Yaskawa INFORM job: FMTV_HOOD_GRILL.JBI

/JOB
//NAME FMTV_HOOD_GRILL
//POS
///NPOS 94,0,0,0,0,0
///TOOL 0
///POSTYPE PULSE
///PULSE
C00000=-47368,-58389,-75463,-75325,82045,-91552
C00001=-47476,-117254,-81462,-92967,88282,-121381
C00002=-47585,-150180,-39020,-110955,95029,-145196
C00003=-23270,-163326,-19972,-112032,80023,-131681
C00004=-25712,-159380,-18293,-113523,79114,-132193
C00005=-33335,-143978,-10206,-123508,65501,-132940
C00006=-42763,-128241,194,-135326,52037,-131772
C00007=-34360,-122011,4195,-131468,51961,-132252
C00008=23040,-127606,-726,-98184,56131,-134608
C00009=54530,-133930,-312,-87484,54655,-130791
C00010=68015,-137434,2378,-86925,51565,-126975
C00011=68015,-137434,2378,-86925,51565,-126975
C00012=70681,-138644,2888,-85845,52080,-126328
C00013=71040,-140703,2447,-86259,52088,-125743
C00014=69846,-144743,783,-88040,51792,-124880
C00015=57718,-148947,-5081,-83684,62309,-128964
C00016=53995,-150636,-6769,-82722,66165,-129759
C00017=48232,-153207,-9364,-79812,75001,-130904
C00018=44695,-155503,-11225,-75321,85283,-131266
C00019=36329,-165923,-20799,-76940,81382,-133395
C00020=32510,-169572,-22983,-79666,80545,-133049
C00021=-44932,-162730,-9861,-129768,80460,-128201
C00022=-46663,-160332,-8884,-130899,79792,-128432
C00023=-49044,-157772,-7071,-132541,79251,-128470
C00024=-34601,-158442,-13610,-121844,79482,-130617
C00025=-34196,-157366,-13562,-121475,79274,-130894
C00026=-74927,-119102,15325,-149774,69260,-130968
C00027=-88106,-120838,19729,-158428,69500,-128950
C00028=-97244,-122496,24507,-164049,70779,-127710
C00029=-62772,-164018,-8236,-136847,75645,-129302
C00030=-22020,-164296,-20741,-110455,80031,-133645
C00031=-23986,-161695,-19560,-112089,79534,-132888
C00032=-25743,-159215,-18122,-113544,79109,-132191
C00033=7628,-162474,-22830,-93471,80813,-134336
C00034=38278,-166162,-20603,-75650,81675,-133226
C00035=48223,-172527,-17821,-220718,66953,-61657
C00036=20447,-173972,-28067,-239715,62384,-67258
C00037=18257,-169178,-23297,-241360,62687,-67091
C00038=19966,-167669,-22486,-240275,62232,-66992
C00039=54812,-127092,1429,-219590,50281,-66184
C00040=53722,-119295,5623,-221586,49019,-65115
C00041=3138,-117684,4029,-257945,62693,-59441
C00042=-54590,-119527,6471,-291312,81310,-61600
C00043=-61303,-121629,6130,-295408,82823,-62492
C00044=-62473,-124760,4446,-296058,82813,-62956
C00045=-61383,-127382,2761,-295300,82324,-63140
C00046=-45291,-158436,-14199,-283363,76411,-66448
C00047=-36803,-168530,-21385,-279249,73403,-67202
C00048=-33637,-169122,-22414,-277154,72885,-67040
C00049=-8268,-168152,-25177,-260735,67443,-65637
C00050=19974,-167686,-22517,-240273,62227,-66989
C00051=27011,-166914,-18516,-232160,63405,-68805
C00052=41789,-166510,-12245,-220087,63923,-71032
C00053=36873,-171047,-15710,-223565,64778,-70981
C00054=-30875,-170872,-20008,-275129,71015,-67437
C00055=-28839,-166908,-10700,-269968,72597,-69697
C00056=-24201,-165834,-10805,-266909,72004,-69362
C00057=15715,-164670,-9145,-238305,67431,-70401
C00058=16294,-164883,-9077,-237836,67450,-70496
C00059=15032,-168908,-9930,-238193,68465,-71268
C00060=-16532,-170220,-12590,-261050,71283,-70207
C00061=-22086,-169030,-11677,-265035,71861,-70073
C00062=-25053,-166420,-10957,-267434,72126,-69490
C00063=-28592,-172919,-21943,-270605,72527,-68220
C00064=22123,-170087,-18028,-234219,65785,-69866
C00065=20623,-164258,-8108,-234618,67125,-70753
C00066=23795,-164163,-6635,-232067,67258,-71214
C00067=37423,-164557,-4674,-225452,64295,-71455
C00068=49664,-167838,-5549,-221136,60772,-72368
C00069=50042,-168090,-5420,-220785,60902,-72462
C00070=48310,-171489,-6267,-221593,61991,-72941
C00071=47370,-171605,-6665,-222333,61921,-72856
C00072=34595,-170073,-7542,-227989,64921,-72953
C00073=21833,-169684,-9235,-234274,67927,-72789
C00074=20032,-169188,-9766,-235757,67758,-72479
C00075=22853,-164534,-7043,-232761,67333,-71170
C00076=19415,-164420,-8530,-235544,67166,-70642
C00077=23719,-173498,-25771,-233839,64304,-68922
C00078=56681,-170652,-7579,-211590,63873,-72674
C00079=53657,-165861,834,-213371,65473,-73133
C00080=55028,-166339,2357,-212686,65788,-74745
C00081=76216,-161231,29355,-196807,75399,-75518
C00082=76318,-160276,31966,-195629,77283,-75776
C00083=75919,-161073,31738,-195883,77558,-75842
C00084=71583,-166800,24804,-195873,73324,-78712
C00085=69455,-168811,22349,-196597,72549,-80310
C00086=67389,-170127,19199,-198092,71648,-80274
C00087=49281,-173575,-1247,-212167,63667,-78545
C00088=49088,-172813,-1584,-212451,63187,-78362
C00089=54651,-166467,2917,-212327,66600,-74972
C00090=59119,-174402,-10513,-209681,64182,-74287
C00091=59119,-174402,-10513,-209681,64182,-74287
C00092=-41638,-117344,-74516,-143224,92250,-82798
C00093=-47368,-58389,-75463,-75325,82045,-91552
//INST
///DATE 2023/03/28 17:51
///ATTR SC,RW
///GROUP1 RB1
NOP
MOVJ C00000 VJ=65.00  //SAW CHANGE
MOVJ C00001 VJ=65.00  //OVER RIB
MOVJ C00002 VJ=65.00  //ROTATE TO SQUARE UP
MOVJ C00003 VJ=65.00  //ABOVE CUT
MOVL C00004 V=30.0  //INTO CUT
MOVL C00005 V=30.0
MOVL C00006 V=30.0  //BOTTOM INSIDE CORNER
MOVL C00007 V=30.0  //END OF ANGLE
MOVL C00008 V=30.0
MOVL C00009 V=30.0
MOVL C00010 V=30.0
MOVC C00011 V=30.0
MOVC C00012 V=30.0
MOVC C00013 V=30.0
MOVC C00014 V=30.0
MOVL C00015 V=30.0
MOVL C00016 V=30.0
MOVL C00017 V=30.0
MOVL C00018 V=30.0
MOVL C00019 V=30.0
MOVL C00020 V=45.0  //AWAY FROM CUT
MOVL C00021 V=65.0  //UP TO CENTER
MOVL C00022 V=15.0
MOVL C00023 V=15.0  //INTO CENTER
MOVL C00024 V=30.0  //RIGHT TOP CORNER CENTER
MOVL C00025 V=30.0
MOVL C00026 V=30.0  //BOTTOM RIGHT CORNER
MOVL C00027 V=30.0
MOVL C00028 V=30.0  //BOTTOM LEFT CORNER
MOVL C00029 V=30.0  //TOP LEFT CORNER
MOVL C00030 V=65.0  //TO TOP RIGHT
MOVL C00031 V=65.0  //UP TO
MOVL C00032 V=15.0  //INTO TOP RIGHT
MOVL C00033 V=15.0
MOVL C00034 V=15.0  //END TOP RIGHT
MOVJ C00035 VJ=65.00  //ROTATE
MOVL C00036 V=65.0  //OVER LEFT GRILL
MOVL C00037 V=65.0  //UP TO
MOVL C00038 V=30.0  //INTO LEFT
MOVL C00039 V=30.0  //TOP OF ANGLE
MOVL C00040 V=30.0  //BOTTOM ANGLE
MOVL C00041 V=30.0
MOVC C00042 V=30.0
MOVC C00043 V=30.0
MOVC C00044 V=30.0
MOVC C00045 V=30.0
MOVL C00046 V=30.0
MOVL C00047 V=30.0
MOVL C00048 V=30.0
MOVL C00049 V=30.0
MOVL C00050 V=30.0  //END
MOVL C00051 V=30.0  //INTO CENTER
MOVL C00052 V=30.0  //END CENTER
MOVL C00053 V=45.0  //AWAY
MOVL C00054 V=65.0  //TO LEFT SIDE
MOVL C00055 V=65.0  //INLINE WITH CUT
MOVL C00056 V=30.0  //INTO LEFT
MOVL C00057 V=30.0
MOVL C00058 V=30.0
MOVL C00059 V=30.0
MOVL C00060 V=30.0
MOVL C00061 V=30.0
MOVL C00062 V=30.0  //END
MOVL C00063 V=65.0  //AWAY
MOVL C00064 V=65.0  //TO CENTER
MOVL C00065 V=65.0  //INLINE
MOVL C00066 V=15.0  //INTO CUT
MOVL C00067 V=30.0
MOVL C00068 V=30.0
MOVL C00069 V=30.0
MOVL C00070 V=30.0
MOVL C00071 V=30.0
MOVL C00072 V=30.0
MOVL C00073 V=30.0
MOVL C00074 V=30.0
MOVL C00075 V=30.0  //END
MOVL C00076 V=65.0  //AWAY
MOVL C00077 V=65.0  //ABOVE
MOVL C00078 V=65.0  //TO RIGHT
MOVL C00079 V=65.0  //INLINE
MOVL C00080 V=15.0  //INTO
MOVL C00081 V=30.0
MOVL C00082 V=30.0
MOVL C00083 V=30.0
MOVL C00084 V=30.0
MOVL C00085 V=30.0
MOVL C00086 V=30.0
MOVL C00087 V=30.0
MOVL C00088 V=30.0
MOVL C00089 V=30.0  //END
MOVL C00090 V=65.0  //AWAY
MOVJ C00091 VJ=65.00
MOVJ C00092 VJ=65.00
MOVJ C00093 VJ=65.00  //3/16 CHANGE
END
